GLOBALCONSTANTS logiBUS_DI (* logiBUS_DI constants *)
  (* Standard: 61499-1; Description: Copyright (c) 2024 HR Agrartechnik GmbH This program and the accompanying materials are made available under the terms of the Eclipse Public License 2.0 which is available at https://www.eclipse.org/legal/epl-2.0/ SPDX-License-Identifier: EPL-2.0 *)
  (* Version 1.0, 2024-01-25, Franz Höpfinger, HR Agrartechnik GmbH *)
  PACKAGE logiBUS::io::DI;
  IMPORT eclipse4diac::core::TypeHash;
  VAR_GLOBAL CONSTANT
    Input_I1 : logiBUS::io::DI::logiBUS_DI_S := (Pin := 1);
    Input_I2 : logiBUS::io::DI::logiBUS_DI_S := (Pin := 2);
    Input_I3 : logiBUS::io::DI::logiBUS_DI_S := (Pin := 3);
    Input_I4 : logiBUS::io::DI::logiBUS_DI_S := (Pin := 4);
    Input_I5 : logiBUS::io::DI::logiBUS_DI_S := (Pin := 5);
    Input_I6 : logiBUS::io::DI::logiBUS_DI_S := (Pin := 6);
    Input_I7 : logiBUS::io::DI::logiBUS_DI_S := (Pin := 7);
    Input_I8 : logiBUS::io::DI::logiBUS_DI_S := (Pin := 8);
    Input_I9 : logiBUS::io::DI::logiBUS_DI_S := (Pin := 9);
    Invalid : logiBUS::io::DI::logiBUS_DI_S := (Pin := 255);
  END_VAR
END_GLOBALCONSTANTS
